# EPICS autosave request: andorApp/Db/shamrock_settings.req
$(P)$(R)Wavelength
$(P)$(R)Grating
$(P)$(R)SlitSize1
$(P)$(R)SlitSize2
$(P)$(R)SlitSize3
$(P)$(R)SlitSize4
